FUNCTION_BLOCK _ETcVnAdaptiveThresholdMethod_TestSuite EXTENDS TcUnit.FB_TestSuite
VAR
END_VAR

TestAddress();
TestClearReference();
TestClone();
TestTypeNameReturnsExpected();
TestIdentifierReturnsExpected();
TestMakeReferenceToFollowsReference();
TestMakeReferenceToUpdatesReference();
TestSize();
TestValueReturnsExpectedAfterInit();
TestValueReturnsExpectedAfterChange();
TestSerializeTypeWith();
TestSerializeWith();
TestTryDeserializeFrom();
TestTryMakeReferenceToFollowsReference();
TestTryMakeReferenceToUpdatesReference();

METHOD PUBLIC TestAddress
VAR
    _type : _ETcVnAdaptiveThresholdMethod(ETcVnAdaptiveThresholdMethod.TCVN_ATM_MEAN);
    notExpected : PVOID := 0;
    actual : PVOID;
END_VAR
TEST('TestAddress');

actual := _type.Address;

AssertFalse(
    Condition := (notExpected = actual),
    Message := 'Type did not return a valid address.'
);

TEST_FINISHED();
END_METHOD

METHOD PUBLIC TestClearReference
VAR
    _type : _ETcVnAdaptiveThresholdMethod(ETcVnAdaptiveThresholdMethod.TCVN_ATM_MEAN);
	target : ETcVnAdaptiveThresholdMethod := ETcVnAdaptiveThresholdMethod.TCVN_ATM_MEAN;
    expected : ETcVnAdaptiveThresholdMethod := ETcVnAdaptiveThresholdMethod.TCVN_ATM_MEAN;
    actual : ETcVnAdaptiveThresholdMethod;
END_VAR
TEST('TestClearReference');

_type.MakeReferenceTo(target);
_type.ClearReference();
target := ETcVnAdaptiveThresholdMethod.TCVN_ATM_GAUSSIAN;

actual := _type.Value;

AssertEquals(
    Expected := expected,
    Actual := actual,
    Message := 'Value continued to follow target.'
);

TEST_FINISHED();
END_METHOD

METHOD PUBLIC TestClone
VAR
    _type : _ETcVnAdaptiveThresholdMethod(ETcVnAdaptiveThresholdMethod.TCVN_ATM_MEAN);
	clone : I_Datatype;
	isValidClone : BOOL;
	compareResult : DINT;
END_VAR
TEST('TestClone');

clone := _type.Clone();

isValidClone := clone <> 0;

IF isValidClone THEN
	compareResult := memcmp(_type.Address, clone.Address, clone.Size);
END_IF

AssertTrue(
	Condition := isValidClone,
	Message := 'Clone did not produce a clone'
);

AssertEquals_DINT(
	Expected := 0,
    Actual := compareResult,
    Message := 'Clone did not return a valid clone.'
);

clone.Dispose();

TEST_FINISHED();
END_METHOD

METHOD PUBLIC TestIdentifierReturnsExpected
VAR
    _type : _ETcVnAdaptiveThresholdMethod(ETcVnAdaptiveThresholdMethod.TCVN_ATM_MEAN);
    expected : STRING := 'ETcVnAdaptiveThresholdMethod';
    actual : STRING;
END_VAR
TEST('TestIdentifierReturnsExpected');

actual := _type.Identifier;

AssertEquals_STRING(
    Expected := expected,
    Actual := actual,
    Message := 'Type did not return correct iec type.'
);

TEST_FINISHED();
END_METHOD

METHOD PUBLIC TestMakeReferenceToFollowsReference
VAR
    _type : _ETcVnAdaptiveThresholdMethod(ETcVnAdaptiveThresholdMethod.TCVN_ATM_MEAN);
	target : ETcVnAdaptiveThresholdMethod := ETcVnAdaptiveThresholdMethod.TCVN_ATM_MEAN;
    expected : ETcVnAdaptiveThresholdMethod := ETcVnAdaptiveThresholdMethod.TCVN_ATM_GAUSSIAN;
    actual : ETcVnAdaptiveThresholdMethod;
END_VAR
TEST('TestMakeReferenceToFollowsReference');

_type.MakeReferenceTo(target);
target := ETcVnAdaptiveThresholdMethod.TCVN_ATM_GAUSSIAN;

actual := _type.Value;

AssertEquals(
    Expected := expected,
    Actual := actual,
    Message := 'Value did not follow target change.'
);

TEST_FINISHED();
END_METHOD

METHOD PUBLIC TestMakeReferenceToUpdatesReference
VAR
    _type : _ETcVnAdaptiveThresholdMethod(ETcVnAdaptiveThresholdMethod.TCVN_ATM_MEAN);
	target : ETcVnAdaptiveThresholdMethod := ETcVnAdaptiveThresholdMethod.TCVN_ATM_MEAN;
    expected : ETcVnAdaptiveThresholdMethod := ETcVnAdaptiveThresholdMethod.TCVN_ATM_GAUSSIAN;
    actual : ETcVnAdaptiveThresholdMethod;
END_VAR
TEST('TestMakeReferenceToUpdatesReference');

_type.MakeReferenceTo(target);
_type.Value := ETcVnAdaptiveThresholdMethod.TCVN_ATM_GAUSSIAN;

actual := target;

AssertEquals(
    Expected := expected,
    Actual := actual,
    Message := 'Value did not update target.'
);

TEST_FINISHED();
END_METHOD

METHOD PUBLIC TestSerializeTypeWith
VAR
    _type : _ETcVnAdaptiveThresholdMethod(ETcVnAdaptiveThresholdMethod.TCVN_ATM_MEAN);
    serializer : JsonSerializer;
    expected : STRING(500) := '{"typeName":"ENUM","identifier":"ETcVnAdaptiveThresholdMethod","enumerations":["TCVN_ATM_MEAN","TCVN_ATM_GAUSSIAN"],"baseType":{"typeName":"DINT","minValue":-2147483648,"maxValue":2147483647,"isSigned":true,"isFloat":false}}'; 
    actual : STRING(500);
END_VAR
TEST('TestSerializeTypeWith');

serializer.Reset();
_type.SerializeTypeWith(serializer);
serializer.TryGetSerializedData(ADR(actual), SIZEOF(actual));

AssertEquals_STRING(
    Expected := expected,
    Actual := actual,
    Message := 'Serialization of type did not return correct string.'
);

TEST_FINISHED();
END_METHOD

METHOD PUBLIC TestSerializeWith
VAR
    _type : _ETcVnAdaptiveThresholdMethod(ETcVnAdaptiveThresholdMethod.TCVN_ATM_MEAN);
    serializer : JsonSerializer;
    expected : STRING := '"TCVN_ATM_MEAN"';
    actual : STRING(500);
END_VAR
TEST('TestSerializeWith');

serializer.Reset();
_type.SerializeWith(serializer);
serializer.TryGetSerializedData(ADR(actual), SIZEOF(actual));

AssertEquals_STRING(
    Expected := expected,
    Actual := actual,
    Message := 'Serialization of type data did not return correct string.'
);

TEST_FINISHED();
END_METHOD

METHOD PUBLIC TestSize
VAR
    _type : _ETcVnAdaptiveThresholdMethod(ETcVnAdaptiveThresholdMethod.TCVN_ATM_MEAN);
    expected : UDINT := SIZEOF(ETcVnAdaptiveThresholdMethod);
    actual : UDINT;
END_VAR
TEST('TestSize');

actual := _type.Size;

AssertEquals_UDINT(
    Expected := Expected,
    Actual := actual,
    Message := 'Type did not return the correct size.'
);

TEST_FINISHED();
END_METHOD

METHOD PUBLIC TestTryDeserializeFrom
VAR
    deserializer : JsonDeserializer;
    feedback : DeserializerFeedback;
    json : STRING := '"TCVN_ATM_MEAN"';
    _type : _ETcVnAdaptiveThresholdMethod(ETcVnAdaptiveThresholdMethod.TCVN_ATM_MEAN);
    expected : ETcVnAdaptiveThresholdMethod := ETcVnAdaptiveThresholdMethod.TCVN_ATM_MEAN;
    actual : ETcVnAdaptiveThresholdMethod;
 END_VAR
TEST('TestTryDeserializeFrom');

deserializer.Reset();
deserializer.TryLoad(json);
_type.TryDeserializeFrom(Deserializer, Feedback);

actual := _type.Value;

AssertEquals(
    Expected := expected,
    Actual := actual,
    Message := 'Type did not deserialize correctly.'
);

TEST_FINISHED();
END_METHOD

METHOD PUBLIC TestTryMakeReferenceToFollowsReference
VAR
    _type : _ETcVnAdaptiveThresholdMethod(ETcVnAdaptiveThresholdMethod.TCVN_ATM_MEAN);
	target : _ETcVnAdaptiveThresholdMethod(ETcVnAdaptiveThresholdMethod.TCVN_ATM_MEAN);
    expected : ETcVnAdaptiveThresholdMethod := ETcVnAdaptiveThresholdMethod.TCVN_ATM_GAUSSIAN;
    actual : ETcVnAdaptiveThresholdMethod;
END_VAR
TEST('TestTryMakeReferenceToFollowsReference');

_type.TryMakeReferenceTo(target);
target.Value := ETcVnAdaptiveThresholdMethod.TCVN_ATM_GAUSSIAN;

actual := _type.Value;

AssertEquals(
    Expected := expected,
    Actual := actual,
    Message := 'Value did not follow target change.'
);

TEST_FINISHED();
END_METHOD

METHOD PUBLIC TestTryMakeReferenceToUpdatesReference
VAR
    _type : _ETcVnAdaptiveThresholdMethod(ETcVnAdaptiveThresholdMethod.TCVN_ATM_MEAN);
	target : _ETcVnAdaptiveThresholdMethod(ETcVnAdaptiveThresholdMethod.TCVN_ATM_MEAN);
    expected : ETcVnAdaptiveThresholdMethod := ETcVnAdaptiveThresholdMethod.TCVN_ATM_GAUSSIAN;
    actual : ETcVnAdaptiveThresholdMethod;
END_VAR
TEST('TestTryMakeReferenceToUpdatesReference');

_type.TryMakeReferenceTo(target);
_type.Value := ETcVnAdaptiveThresholdMethod.TCVN_ATM_GAUSSIAN;

actual := target.Value;

AssertEquals(
    Expected := expected,
    Actual := actual,
    Message := 'Value did not update target.'
);

TEST_FINISHED();
END_METHOD

METHOD PUBLIC TestTypeNameReturnsExpected
VAR
    _type : _ETcVnAdaptiveThresholdMethod(ETcVnAdaptiveThresholdMethod.TCVN_ATM_MEAN);
    expected : STRING := 'ENUM';
    actual : STRING;
END_VAR
TEST('TestTypeNameReturnsExpected');

actual := _type.TypeName;

AssertEquals_STRING(
    Expected := expected,
    Actual := actual,
    Message := 'Type did not return correct iec type.'
);

TEST_FINISHED();
END_METHOD

METHOD PUBLIC TestValueReturnsExpectedAfterChange
VAR
    _type : _ETcVnAdaptiveThresholdMethod(ETcVnAdaptiveThresholdMethod.TCVN_ATM_MEAN);
    expected : ETcVnAdaptiveThresholdMethod := ETcVnAdaptiveThresholdMethod.TCVN_ATM_GAUSSIAN;
    actual : ETcVnAdaptiveThresholdMethod;
END_VAR
TEST('TestValueReturnsExpectedAfterChange');

_type.Value := ETcVnAdaptiveThresholdMethod.TCVN_ATM_GAUSSIAN;

actual := _type.Value;

AssertEquals(
    Expected := expected,
    Actual := actual,
    Message := 'Expected value not returned after change.'
);

TEST_FINISHED();
END_METHOD

METHOD PUBLIC TestValueReturnsExpectedAfterInit
VAR
    _type : _ETcVnAdaptiveThresholdMethod(ETcVnAdaptiveThresholdMethod.TCVN_ATM_MEAN);
    expected : ETcVnAdaptiveThresholdMethod := ETcVnAdaptiveThresholdMethod.TCVN_ATM_MEAN;
    actual : ETcVnAdaptiveThresholdMethod;
END_VAR
TEST('TestValueReturnsExpectedAfterInit');

actual := _type.Value;

AssertEquals(
    Expected := expected,
    Actual := actual,
    Message := 'Expected value not returned after Init.'
);

TEST_FINISHED();
END_METHOD

END_FUNCTION_BLOCK

(* stored: Version 1.1.0.1, ProductVersion 3.1.4024.12
   POU _ETcVnAdaptiveThresholdMethod_TestSuite: Id {e6a46894-7ca9-097b-2563-300c3b385bcd}, SpecialFunc None
   Method TestAddress: Id {f9f3a4ca-c47d-0952-2180-19eb659a5b31}
   Method TestClearReference: Id {ff05fdcc-f901-03f9-3e4e-0312520ac416}
   Method TestClone: Id {eac501f6-cc4c-0279-0bf7-c7d37bbbbd7a}
   Method TestIdentifierReturnsExpected: Id {4ca99e80-19d9-043b-0a90-8f87186069aa}
   Method TestMakeReferenceToFollowsReference: Id {3c6c916b-0015-0d37-14f0-35dd8f8b2319}
   Method TestMakeReferenceToUpdatesReference: Id {46c8fd8e-640c-0b39-0aca-c0c98f31fcbd}
   Method TestSerializeTypeWith: Id {61495043-845d-02be-323a-4b6f7fe06b9b}
   Method TestSerializeWith: Id {1cc8290e-bbfe-0f9a-12e8-453b42f1408c}
   Method TestSize: Id {9c3ee854-9ce2-012d-0bf9-47fc26acfcad}
   Method TestTryDeserializeFrom: Id {340455b2-e36e-01b2-3e53-28c50f7283e5}
   Method TestTryMakeReferenceToFollowsReference: Id {b696cc68-a552-0318-09c3-d16ebfaa510c}
   Method TestTryMakeReferenceToUpdatesReference: Id {5ec96838-aaa8-0d36-3b68-eb363f22a428}
   Method TestTypeNameReturnsExpected: Id {e1760cdf-6d13-0bed-075e-ad99dba075bb}
   Method TestValueReturnsExpectedAfterChange: Id {d8dd6afb-65fa-07a9-02db-2361a3024fd5}
   Method TestValueReturnsExpectedAfterInit: Id {c4b5fa1a-5ede-0af2-287b-0cf56ad80ef3} *)
